PROGRAM MainTestPart
VAR
	//**************************write data to file or read data from file****************************//
	m_FB_CSV_TextMode_ReadWrite1:FB_CSV_TextMode_ReadWrite;	
	m_bWrite: BOOL;
	m_writedata:ARRAY[0..19,0..9] OF LREAL;
	m_bRead:BOOL;
	m_readdata:ARRAY[0..10000,0..120] OF LREAL;
	
	
	
	
	//**********************************single arm test related data****************************//
	m_armSelect:INT:=1;
	m_writeStart:BOOL;
	m_writeFinished:BOOL;
	m_writeStep:INT:=-1;
	m_fileId:INT;
	sFileName:T_MaxString;
	
	//data
	m_time:LREAL;
	m_row,m_col:INT;
	m_testDataWriteEnable:BOOL;	
	
	(*
	m_jntTrqD2,m_jntTrqD3:ARRAY[0..(gvl_const.g_writeDataNum-1),0..6] OF LREAL;
	m_jntPosD2,m_jntPosD3:ARRAY[0..(gvl_const.g_writeDataNum-1),0..6] OF LREAL;
	m_cmdDHjntPosD2,m_cmdDHjntPosD3:ARRAY[0..(gvl_const.g_writeDataNum-1),0..6] OF LREAL;
	m_data:ARRAY[0..(gvl_const.g_writeDataNum-1),0..6] OF LREAL;
	
	//pointer to global variables
	g_pcmdDHJntPosD2,g_pJntPosD2,g_pJntTrqD2:POINTER TO ARRAY[1..g_mArmNum,1..g_mJntNum,1..gvl_const.g_recordDataNum] OF LREAL;
	g_pcmdDHJntPosD3,g_pJntPosD3,g_pJntTrqD3:POINTER TO ARRAY[1..g_mArmNum,1..g_mJntNum,1..gvl_const.g_recordDataNum] OF LREAL;
	
	//data from global variables
	m_cmdDHJntPosD2_data,m_JntPosD2_data,m_JntTrqD2_data:ARRAY[1..g_mArmNum,1..g_mJntNum,1..gvl_const.g_recordDataNum] OF LREAL;
	m_cmdDHJntPosD3_data,m_JntPosD3_data,m_JntTrqD3_data:ARRAY[1..g_mArmNum,1..g_mJntNum,1..gvl_const.g_recordDataNum] OF LREAL;
	*)
	
	
	
	
	//**********************************write precision test data**********************************//
	m_armMatId:INT:=1;
	m_matWriteStep:INT:=-1;
	m_matrixData:ARRAY[0..3,0..3] OF LREAL;
	m_frontPose:ST_Frame;	
END_VAR

//write the data to file example
dataWriteExp();

//HMI for accuracy test
HmiMid();

//write data related to precision test
writePrecisionData();

METHOD dataWriteExp : BOOL
VAR_INPUT
END_VAR

(*
m_FB_CSV_TextMode_ReadWrite1(	sNetId:= '', 	sFileName:='D:\file20241213.csv' , 	bBusy=> , 	bError=> , 	nErrorID=> , 	nErrorState=> );

m_FB_CSV_TextMode_ReadWrite1.M_WriteCsv(	bExecute:=m_bWrite , 	nMode:= FOPEN_MODEWRITE OR FOPEN_MODETEXT, 
	ptPointer:=ADR(m_writedata) , 	nRows:= 19, 	nColumns:=9 );

m_FB_CSV_TextMode_ReadWrite1.M_ReadCsv(bExecute:=m_bRead , ptPointer:= ADR(m_readdata), nRows:=10000 , nColumns:= 120);
IF NOT m_FB_CSV_TextMode_ReadWrite1.bBusy THEN
	m_bWrite:=FALSE;
	m_bRead:=FALSE;
END_IF
*)
END_METHOD

METHOD HmiMid : BOOL
VAR_INPUT
END_VAR
VAR
	I : INT;
	iArm : INT;
	armId:INT;
END_VAR


//the interface relate to variable A1_Arm1Mode
FOR I:=1 TO 4  DO
	FOR iARM:=1 TO gvl_accuracyTest.g_controlModeNum DO 
		//Monitoring button signal rising edge
		A1_Arm1Mode_TRIG[i,iARM](CLK:=A1_Arm1Mode[I,iARM],Q=>);
		IF A1_Arm1Mode_TRIG[i,iARM].Q THEN 
			A1_Arm1Mode:=A1_Arm1Mode_Mid;
			GVL_AccuracyTestVar.g_controlMode[i]:=iARM;
			A1_Arm1Mode[i,iARM]:=TRUE;
		END_IF		
		
		//Monitoring button signal falling edge
		A1_Arm1Mode_F_TRIG[i,iARM](CLK:=A1_Arm1Mode[I,iARM]);		
	END_FOR
	
	//If a signal falling edge is detected,Set variables to default values---continuous joint motion or continuous space motion
	IF A1_Arm1Mode_F_TRIG[i,2].Q OR A1_Arm1Mode_F_TRIG[i,4].Q THEN
		GVL_AccuracyTestVar.g_controlMode[i]:=0;
		A1_Arm1Mode:=A1_Arm1Mode_Mid;
	END_IF
	
	//If the accuracy test or workspace test is in progress, click the return to origin button to exit the accuracy test
	IF (GVL_AccuracyTestVar.g_controlMode[i]=5) THEN
		IF (A1_Arm1Mode[i,6]=TRUE) THEN
			GVL_AccuracyTestVar.g_controlMode[i]:=0;
			A1_Arm1Mode:=A1_Arm1Mode_Mid;
		END_IF
	END_IF
END_FOR


//Upload variables for displaying button colors
A1_Arm1ModeL:=A1_Arm1Mode_Mid;
A1_Arm1ModeL[1,GVL_AccuracyTestVar.g_controlMode[1]]:=TRUE;
A1_Arm1ModeL[2,GVL_AccuracyTestVar.g_controlMode[2]]:=TRUE;
A1_Arm1ModeL[3,GVL_AccuracyTestVar.g_controlMode[3]]:=TRUE;
A1_Arm1ModeL[4,GVL_AccuracyTestVar.g_controlMode[4]]:=TRUE;


//If the motion ends, set the relevant variables to false
FOR i:=1 TO 4  DO
	IF GVL_AccuracyTestVar.g_controlMode[i]<>0 THEN
		GVL_AccuracyTestVar.g_startMotion[i]:=TRUE;
	ELSE
		GVL_AccuracyTestVar.g_startMotion[i]:=FALSE;
	END_IF
END_FOR


//ui signal copy
GVL_AccuracyTestVar.g_uiArmMode:=A1_Arm1Mode;
END_METHOD

METHOD writePrecisionData : BOOL
VAR_INPUT
	
END_VAR
VAR
	i,j:INT;
END_VAR


FOR i:=1 TO 4 BY 1 DO
	IF (gvl_AccuracyTestVar.g_writeData[i]=TRUE) THEN
		gvl_AccuracyTestVar.g_writeData[i]:=FALSE;
		m_armMatId:=i;
		m_matWriteStep:=0;
	END_IF
END_FOR


CASE m_matWriteStep OF
	0: //prepare for the data
		m_frontPose:=gvl_AccuracyTestVar.g_frontPose[m_armMatId];
		FOR i:=1 TO 3 BY 1 DO			
			FOR j:=1 TO 3 BY 1 DO
				m_matrixData[i-1,j-1]:=m_frontPose.m_rot[i,j];
			END_FOR
		END_FOR
		
		FOR i:=1 TO 3 BY 1 DO
			m_matrixData[i-1,4-1]:=m_frontPose.m_pos[i];
		END_FOR
		m_matWriteStep:=10;
		
		
	10:
		IF (m_armMatId=1) THEN
			sFileName:='D:\arm1.txt';
		ELSIF (m_armMatId=2) THEN
			sFileName:='D:\arm2.txt';
		ELSIF (m_armMatId=3) THEN
			sFileName:='D:\arm3.txt';
		ELSIF (m_armMatId=4) THEN
			sFileName:='D:\arm4.txt';
		END_IF
		
		m_row:=3;
		m_col:=3;
		m_time:=0;
		m_matWriteStep:=20;
		
		
	20: //write the joint position
		m_FB_CSV_TextMode_ReadWrite1(	sNetId:= '', 	sFileName:=sFileName , 	bBusy=> , 	bError=> , 	nErrorID=> , 	nErrorState=> );
		m_FB_CSV_TextMode_ReadWrite1.M_WriteCsv(	bExecute:=TRUE , 	nMode:= FOPEN_MODEWRITE OR FOPEN_MODETEXT, 
			ptPointer:=ADR(m_matrixData) , 	nRows:= INT_TO_UINT(m_row), 	nColumns:=INT_TO_UINT(m_col) );
			
		//timer
		m_time:=m_time+0.010;
		
		IF (NOT m_FB_CSV_TextMode_ReadWrite1.bBusy) THEN
			m_FB_CSV_TextMode_ReadWrite1.M_WriteCsv(	bExecute:=FALSE , 	nMode:= FOPEN_MODEWRITE OR FOPEN_MODETEXT, 
			ptPointer:=ADR(m_matrixData) , 	nRows:= INT_TO_UINT(m_row), 	nColumns:=INT_TO_UINT(m_col) );
			m_matWriteStep:=30;
			m_time:=0;
		END_IF
	
	
	30: //end
		m_matWriteStep:=-1;

		
	-1: //
END_CASE
END_METHOD

END_PROGRAM

(* stored: Version 1.1.0.1, ProductVersion 3.1.4024.11
   POU MainTestPart: Id {b83618ba-430f-4dc7-b8e8-725dcbac1ae2}, SpecialFunc None
   Method dataWriteExp: Id {83e2b061-240b-48f5-a37e-40e2d8eb7275}
   Method HmiMid: Id {9a887a90-c99e-4390-abdb-ad0ecd202ca8}
   Method writePrecisionData: Id {029cd9d3-0755-4d4e-9858-76805cdd3ded} *)
